(* IEC 61131-3 sources: uniset2/extensions/JScript/examples, 2 files *)

(* ---- hvac.st ---- *)
(* HVAC Controller — two-zone heating/cooling with alarms
 *
 * Zone 1: Office — heating only
 * Zone 2: Server room — cooling only
 * Common: outdoor temperature sensor, alarm system
 *)

TYPE ZoneConfig :
STRUCT
    setpoint : REAL := 22.0;
    hysteresis : REAL := 1.5;
    alarmHigh : REAL := 35.0;
    alarmLow : REAL := 5.0;
END_STRUCT
END_TYPE

PROGRAM HVAC
VAR_INPUT
    OutdoorTemp : REAL;
    Zone1Temp : REAL;
    Zone2Temp : REAL;
    Enable : BOOL;
    Reset : BOOL;
    ManualMode : BOOL;
END_VAR
VAR_OUTPUT
    Zone1Heater : BOOL;
    Zone2Cooler : BOOL;
    AlarmZone1 : BOOL;
    AlarmZone2 : BOOL;
    AlarmCommon : BOOL;
    RunHours : INT;
END_VAR
VAR
    cfgZone1 : ZoneConfig;
    cfgZone2 : ZoneConfig;
    enableEdge : R_TRIG;
    resetEdge : R_TRIG;

    (* Zone 1: heating *)
    z1_hyst : HYSTERESIS;
    z1_onDelay : TON;
    z1_offDelay : TOF;
    z1_alarmHigh : LIMITALARM;
    z1_cycles : CTU;

    (* Zone 2: cooling *)
    z2_hyst : HYSTERESIS;
    z2_onDelay : TON;
    z2_offDelay : TOF;
    z2_alarmHigh : LIMITALARM;
    z2_cycles : CTU;

    (* Common *)
    blinker : BLINK;
    runTimer : TON;
    runCounter : CTU;
    state : INT := 0;
END_VAR

(* Enable/Reset edge detection *)
enableEdge(CLK := Enable);
resetEdge(CLK := Reset);

IF enableEdge.Q THEN
    state := 1;
END_IF;

IF resetEdge.Q THEN
    state := 0;
    AlarmZone1 := FALSE;
    AlarmZone2 := FALSE;
    AlarmCommon := FALSE;
END_IF;

CASE state OF
    0: (* Standby *)
        Zone1Heater := FALSE;
        Zone2Cooler := FALSE;

    1: (* Running *)
        IF NOT ManualMode THEN
            (* Zone 1: Heating — turn on below setpoint-hyst, off above setpoint+hyst *)
            z1_hyst(IN := Zone1Temp, HIGH := cfgZone1.setpoint + cfgZone1.hysteresis,
                    LOW := cfgZone1.setpoint - cfgZone1.hysteresis);
            z1_onDelay(IN := z1_hyst.OUT, PT := T#3s);
            z1_offDelay(IN := z1_onDelay.Q, PT := T#10s);
            Zone1Heater := z1_offDelay.Q;

            (* Zone 2: Cooling — turn on above setpoint+hyst, off below setpoint-hyst *)
            z2_hyst(IN := Zone2Temp, HIGH := cfgZone2.setpoint + cfgZone2.hysteresis,
                    LOW := cfgZone2.setpoint - cfgZone2.hysteresis);
            z2_onDelay(IN := NOT z2_hyst.OUT, PT := T#5s);
            z2_offDelay(IN := z2_onDelay.Q, PT := T#15s);
            Zone2Cooler := z2_offDelay.Q;
        END_IF;

        (* Alarm monitoring *)
        z1_alarmHigh(IN := Zone1Temp, HIGH := cfgZone1.alarmHigh, LOW := cfgZone1.alarmLow);
        z2_alarmHigh(IN := Zone2Temp, HIGH := cfgZone2.alarmHigh, LOW := cfgZone2.alarmLow);

        AlarmZone1 := NOT z1_alarmHigh.IL;
        AlarmZone2 := NOT z2_alarmHigh.IL;

        IF AlarmZone1 OR AlarmZone2 THEN
            AlarmCommon := TRUE;
            blinker(ENABLE := TRUE, TIMEHIGH := T#500ms, TIMELOW := T#500ms);
        ELSE
            blinker(ENABLE := FALSE, TIMEHIGH := T#500ms, TIMELOW := T#500ms);
        END_IF;

        (* Run hours counter *)
        runTimer(IN := TRUE, PT := T#60s);
        z1_cycles(CU := z1_onDelay.Q, RESET := Reset, PV := 1000);
        z2_cycles(CU := z2_onDelay.Q, RESET := Reset, PV := 1000);
        runCounter(CU := runTimer.Q, RESET := Reset, PV := 10000);
        RunHours := runCounter.CV;

    2: (* Fault *)
        Zone1Heater := FALSE;
        Zone2Cooler := FALSE;
END_CASE;

END_PROGRAM

(* ---- thermostat.st ---- *)
(* Thermostat controller example
 *
 * Demonstrates:
 * - STRUCT type for configuration
 * - State machine (CASE)
 * - Hysteresis control
 * - Standard FBs: R_TRIG, TON, TOF, CTU
 * - Alarm monitoring
 *
 * Convert to JS:
 *   uniset2-st2js thermostat.st -m thermostat_mapping.yaml --debug -o main-plc.js
 *
 * Run with debug:
 *   uniset2-jscript --js-file main-plc.js --confile test.xml --js-name TestProc --js-confnode JSProxy
 *   Open http://host:8088/debug/ui in browser
 *)

TYPE TempConfig :
STRUCT
    setpoint : REAL := 20.0;
    hysteresis : REAL := 2.0;
    maxTemp : REAL := 95.0;
END_STRUCT
END_TYPE

PROGRAM Thermostat
VAR_INPUT
    CurrentTemp : REAL;
    Enable : BOOL;
    Reset : BOOL;
END_VAR
VAR_OUTPUT
    HeaterOn : BOOL;
    AlarmHigh : BOOL;
    CycleCount : INT;
END_VAR
VAR
    config : TempConfig;
    onDelay : TON;
    offDelay : TOF;
    startEdge : R_TRIG;
    cycleCounter : CTU;
    state : INT := 0;    (* 0=Idle, 1=Running, 2=Alarm *)
END_VAR

(* Detect enable button rising edge *)
startEdge(CLK := Enable);
IF startEdge.Q THEN
    state := 1;
END_IF;

(* State machine *)
CASE state OF
    0: (* Idle — heater off *)
        HeaterOn := FALSE;

    1: (* Running — hysteresis control *)
        IF CurrentTemp < config.setpoint - config.hysteresis THEN
            HeaterOn := TRUE;
        ELSIF CurrentTemp > config.setpoint + config.hysteresis THEN
            HeaterOn := FALSE;
        END_IF;

        (* Count heater-on cycles via on-delay *)
        onDelay(IN := HeaterOn, PT := T#5s);
        cycleCounter(CU := onDelay.Q, RESET := Reset, PV := 100);
        CycleCount := cycleCounter.CV;

    2: (* Alarm — emergency stop *)
        HeaterOn := FALSE;
END_CASE;

(* Overtemperature alarm *)
IF CurrentTemp > config.maxTemp THEN
    AlarmHigh := TRUE;
    state := 2;
END_IF;

(* Reset from alarm *)
IF Reset THEN
    state := 0;
    AlarmHigh := FALSE;
END_IF;

END_PROGRAM
